// TIA Portal V20 export
DATA_BLOCK "InstLimitValueDataset1"   // DB54
TITLE = Instance LimitValueDataset1
{ DB_Accessible_From_OPC_UA := 'FALSE' }
AUTHOR : SICAR
FAMILY : ProdData
// Instance DB
// stored: DBAccessibleFromOPCUA false, InstanceOfName LSicar_ProdDataLimitValues, InstanceOfType FB
"LSicar_ProdDataLimitValues"
   // VAR_INPUT
   //    numberConfigDataSets { ExternalAccessible := 'False'; ExternalVisible := 'False'; ExternalWritable := 'False'} : Int;
   //    dataSetNumber { ExternalAccessible := 'False'; ExternalVisible := 'False'; ExternalWritable := 'False'} : UInt;
   // END_VAR
   // VAR_IN_OUT
   //    numberOfDataSets : "LSicar_typeNumberOfDataSets";
   //    dataSet : "LSicar_typeLimitValue";
   //    colorCodeSelectButton { ExternalAccessible := 'False'; ExternalVisible := 'False'; ExternalWritable := 'False'} : UInt;
   // END_VAR
   // VAR
   //    statLimitValue { ExternalAccessible := 'False'; ExternalVisible := 'False'; ExternalWritable := 'False'} : Array[0..10] of "LSicar_typeEdgePulseStruct";
   //    statPrewarnActive { ExternalAccessible := 'False'; ExternalVisible := 'False'; ExternalWritable := 'False'} : Bool;
   //    statAlarmActive { ExternalAccessible := 'False'; ExternalVisible := 'False'; ExternalWritable := 'False'} : Bool;
   // END_VAR
BEGIN
END_DATA_BLOCK
